TYPE ST_LaudaWriteCommands :
STRUCT
	Temperature			: ST_LaudaWriteCommands_Temperature;
	Control				: ST_LaudaWriteCommands_Control;
	ControlParameters	: ST_LaudaWriteCommands_ControlParameters;
	Cooling				: ST_LaudaWriteCommands_Cooling;
	Pump				: ST_LaudaWriteCommands_Pump;
	Rights				: ST_LaudaWriteCommands_Rights;
	Safety				: ST_LaudaWriteCommands_Safety;
	Status				: ST_LaudaWriteCommands_Status;
END_STRUCT
END_TYPE

(* stored: Version 1.1.0.1, ProductVersion 3.1.4024.13
   DUT ST_LaudaWriteCommands: Id {5609a9c4-6754-4c05-80b2-98fed905fa83} *)
